(* Logix 5000 project; controller CHASKEY Emulate 5570 rev 30.12; software revision 30.00 *)

TASK MainTask (periodic, rate 3000 ms, priority 1, watchdog 5000 ms) : MainProgram

MODULES
   Local : Emulate 5570 (ICP 2, rev 30.12)
END_MODULES

VAR_GLOBAL   (* controller tags *)
   _SEC_P : BOOL;
   done : DINT;
   R_TRIG : FBD_ONESHOT;
   temp_var : DINT;
   test_array : DINT[20] := ([0] := 1, [1] := 2, [2] := 3, [3] := 4, [4] := 5, [5] := 6, [6] := 7, [7] := 8, [8] := 9, [9] := 10, [10] := 11, [11] := 12, [12] := 13, [13] := 14, [14] := 15, [15] := 16, [16] := 17, [17] := 18, [18] := 19, [19] := 20);
   TON : FBD_TIMER;
END_VAR

PROGRAM MainProgram   (* main routine MainRoutine *)
VAR
   Chaskey_128_i : DINT;
   Chaskey_a : DINT; {access None}
   Chaskey_BNum : DINT; {access None}
   Chaskey_i : DINT; {access None}
   Chaskey_IndexDiv : DINT;
   Chaskey_IndexMod : DINT;
   Chaskey_input_pi : DINT[4]; {access None}
   Chaskey_j : DINT; {access None}
   Chaskey_key : DINT[4]; {access None}
   Chaskey_L : DINT[4]; {access None}
   Chaskey_LastBlk : DINT[4];
   Chaskey_lb : DINT[16];
   Chaskey_Message : DINT[256]; {access None}
   Chaskey_mlen : DINT;
   Chaskey_MsgBitLen : DINT; {access None}
   Chaskey_MsgBlk : DINT[64];
   Chaskey_MsgBlkLen : DINT;
   Chaskey_per_i : DINT; {access None}
   Chaskey_round : DINT;
   Chaskey_subkey1_i : DINT; {access None}
   Chaskey_subkey2_i : DINT; {access None}
   Chaskey_subkey_1 : DINT[8];
   Chaskey_subkey_2 : DINT[8]; {access None}
   Chaskey_tag : DINT[4]; {access None}
   Chaskey_Temp : DINT; {access None}
   Chaskey_z : DINT;
   SCAN_CYCLE_TIME : DINT; {access None}
   test_i : DINT;
END_VAR

ROUTINE CHASKEY_128   (* structured text *)
   JSR(CHASKEY_Init);
   
   Chaskey_BNum:= Chaskey_MsgBitLen/128;
   
   if Chaskey_MsgBitLen mod 128 <>0 then
   	Chaskey_BNum:= Chaskey_BNum+1;
   end_if;
   
   
   for Chaskey_i:=0 to Chaskey_mlen by 1 do
   	Chaskey_MsgBlkLen:=Chaskey_mlen/4;
   	Chaskey_z:=Chaskey_i mod 4;
   	for Chaskey_j:=0 to 7 by 1 do
   		Chaskey_MsgBlk[Chaskey_MsgBlkLen].[Chaskey_z*8+Chaskey_j]:=Chaskey_Message[Chaskey_i].[Chaskey_j];
   	end_for;
   end_for;
   
   Chaskey_input_pi[3] := Chaskey_key[3];
   Chaskey_input_pi[2] := Chaskey_key[2] ;
   Chaskey_input_pi[1] := Chaskey_key[1] ;
   Chaskey_input_pi[0] := Chaskey_key[0] ;
   
   Chaskey_i:=0;
   if Chaskey_mlen<>0 then
   	while Chaskey_i < Chaskey_BNum-1 do
   		Chaskey_128_i:=Chaskey_i*4;
   		Chaskey_input_pi[3] := Chaskey_input_pi[3] XOR Chaskey_MsgBlk[Chaskey_128_i+3];
   		Chaskey_input_pi[2] := Chaskey_input_pi[2] XOR Chaskey_MsgBlk[Chaskey_128_i+2];
   		Chaskey_input_pi[1] := Chaskey_input_pi[1] XOR Chaskey_MsgBlk[Chaskey_128_i+1];
   		Chaskey_input_pi[0] := Chaskey_input_pi[0] XOR Chaskey_MsgBlk[Chaskey_128_i+0];
   		JSR(CHASKEY_Permutation);
   
   		if Chaskey_i>=Chaskey_BNum-2 then
   			Exit;
   		end_if;
   
   		Chaskey_i:=Chaskey_i +1;
   	end_while;
   end_if;
   
   
   if (Chaskey_mlen<>0) AND ((Chaskey_mlen & 15)=0) then
   	Chaskey_L[3] := Chaskey_subkey_1[3];
   	Chaskey_L[2] := Chaskey_subkey_1[2] ;
   	Chaskey_L[1] := Chaskey_subkey_1[1] ;
   	Chaskey_L[0] := Chaskey_subkey_1[0] ;
   	Chaskey_LastBlk[0]:=Chaskey_MsgBlk[0];
   	Chaskey_LastBlk[1]:=Chaskey_MsgBlk[1];
   	Chaskey_LastBlk[2]:=Chaskey_MsgBlk[2];
   	Chaskey_LastBlk[3]:=Chaskey_MsgBlk[3];
   else
   	Chaskey_L[3] := Chaskey_subkey_2[3];
   	Chaskey_L[2] := Chaskey_subkey_2[2] ;
   	Chaskey_L[1] := Chaskey_subkey_2[1] ;
   	Chaskey_L[0] := Chaskey_subkey_2[0] ;
   
   
   	Chaskey_IndexMod:= Chaskey_mlen mod 16;
   	Chaskey_IndexDiv:= (Chaskey_mlen/16)*16;
   	for Chaskey_j:=0 to Chaskey_IndexMod-1 by 1 do
   		Chaskey_lb[Chaskey_j]:=Chaskey_Message[Chaskey_IndexDiv+Chaskey_j];
   	end_for;
   	Chaskey_lb[Chaskey_IndexMod]:=1;
   	for Chaskey_j:=Chaskey_IndexMod+1 to 15 by 1 do
   		Chaskey_lb[Chaskey_j]:=0;
   	end_for;
   
   	//lastblock = (uint32_t*) lb;
   	Chaskey_LastBlk[0].0:=Chaskey_lb[0].0;
   	Chaskey_LastBlk[0].1:=Chaskey_lb[0].1;
   	Chaskey_LastBlk[0].2:=Chaskey_lb[0].2;
   	Chaskey_LastBlk[0].3:=Chaskey_lb[0].3;
   	Chaskey_LastBlk[0].4:=Chaskey_lb[0].4;
   	Chaskey_LastBlk[0].5:=Chaskey_lb[0].5;
   	Chaskey_LastBlk[0].6:=Chaskey_lb[0].6;
   	Chaskey_LastBlk[0].7:=Chaskey_lb[0].7;
   	Chaskey_LastBlk[0].8:=Chaskey_lb[1].0;
   	Chaskey_LastBlk[0].9:=Chaskey_lb[1].1;
   	Chaskey_LastBlk[0].10:=Chaskey_lb[1].2;
   	Chaskey_LastBlk[0].11:=Chaskey_lb[1].3;
   	Chaskey_LastBlk[0].12:=Chaskey_lb[1].4;
   	Chaskey_LastBlk[0].13:=Chaskey_lb[1].5;
   	Chaskey_LastBlk[0].14:=Chaskey_lb[1].6;
   	Chaskey_LastBlk[0].15:=Chaskey_lb[1].7;
   	Chaskey_LastBlk[0].16:=Chaskey_lb[2].0;
   	Chaskey_LastBlk[0].17:=Chaskey_lb[2].1;
   	Chaskey_LastBlk[0].18:=Chaskey_lb[2].2;
   	Chaskey_LastBlk[0].19:=Chaskey_lb[2].3;
   	Chaskey_LastBlk[0].20:=Chaskey_lb[2].4;
   	Chaskey_LastBlk[0].21:=Chaskey_lb[2].5;
   	Chaskey_LastBlk[0].22:=Chaskey_lb[2].6;
   	Chaskey_LastBlk[0].23:=Chaskey_lb[2].7;
   	Chaskey_LastBlk[0].24:=Chaskey_lb[3].0;
   	Chaskey_LastBlk[0].25:=Chaskey_lb[3].1;
   	Chaskey_LastBlk[0].26:=Chaskey_lb[3].2;
   	Chaskey_LastBlk[0].27:=Chaskey_lb[3].3;
   	Chaskey_LastBlk[0].28:=Chaskey_lb[3].4;
   	Chaskey_LastBlk[0].29:=Chaskey_lb[3].5;
   	Chaskey_LastBlk[0].30:=Chaskey_lb[3].6;
   	Chaskey_LastBlk[0].31:=Chaskey_lb[3].7;
   
   	Chaskey_LastBlk[1].0:=Chaskey_lb[4].0;
   	Chaskey_LastBlk[1].1:=Chaskey_lb[4].1;
   	Chaskey_LastBlk[1].2:=Chaskey_lb[4].2;
   	Chaskey_LastBlk[1].3:=Chaskey_lb[4].3;
   	Chaskey_LastBlk[1].4:=Chaskey_lb[4].4;
   	Chaskey_LastBlk[1].5:=Chaskey_lb[4].5;
   	Chaskey_LastBlk[1].6:=Chaskey_lb[4].6;
   	Chaskey_LastBlk[1].7:=Chaskey_lb[4].7;
   	Chaskey_LastBlk[1].8:=Chaskey_lb[5].0;
   	Chaskey_LastBlk[1].9:=Chaskey_lb[5].1;
   	Chaskey_LastBlk[1].10:=Chaskey_lb[5].2;
   	Chaskey_LastBlk[1].11:=Chaskey_lb[5].3;
   	Chaskey_LastBlk[1].12:=Chaskey_lb[5].4;
   	Chaskey_LastBlk[1].13:=Chaskey_lb[5].5;
   	Chaskey_LastBlk[1].14:=Chaskey_lb[5].6;
   	Chaskey_LastBlk[1].15:=Chaskey_lb[5].7;
   	Chaskey_LastBlk[1].16:=Chaskey_lb[6].0;
   	Chaskey_LastBlk[1].17:=Chaskey_lb[6].1;
   	Chaskey_LastBlk[1].18:=Chaskey_lb[6].2;
   	Chaskey_LastBlk[1].19:=Chaskey_lb[6].3;
   	Chaskey_LastBlk[1].20:=Chaskey_lb[6].4;
   	Chaskey_LastBlk[1].21:=Chaskey_lb[6].5;
   	Chaskey_LastBlk[1].22:=Chaskey_lb[6].6;
   	Chaskey_LastBlk[1].23:=Chaskey_lb[6].7;
   	Chaskey_LastBlk[1].24:=Chaskey_lb[7].0;
   	Chaskey_LastBlk[1].25:=Chaskey_lb[7].1;
   	Chaskey_LastBlk[1].26:=Chaskey_lb[7].2;
   	Chaskey_LastBlk[1].27:=Chaskey_lb[7].3;
   	Chaskey_LastBlk[1].28:=Chaskey_lb[7].4;
   	Chaskey_LastBlk[1].29:=Chaskey_lb[7].5;
   	Chaskey_LastBlk[1].30:=Chaskey_lb[7].6;
   	Chaskey_LastBlk[1].31:=Chaskey_lb[7].7;
   
   	Chaskey_LastBlk[2].0:=Chaskey_lb[8].0;
   	Chaskey_LastBlk[2].1:=Chaskey_lb[8].1;
   	Chaskey_LastBlk[2].2:=Chaskey_lb[8].2;
   	Chaskey_LastBlk[2].3:=Chaskey_lb[8].3;
   	Chaskey_LastBlk[2].4:=Chaskey_lb[8].4;
   	Chaskey_LastBlk[2].5:=Chaskey_lb[8].5;
   	Chaskey_LastBlk[2].6:=Chaskey_lb[8].6;
   	Chaskey_LastBlk[2].7:=Chaskey_lb[8].7;
   	Chaskey_LastBlk[2].8:=Chaskey_lb[9].0;
   	Chaskey_LastBlk[2].9:=Chaskey_lb[9].1;
   	Chaskey_LastBlk[2].10:=Chaskey_lb[9].2;
   	Chaskey_LastBlk[2].11:=Chaskey_lb[9].3;
   	Chaskey_LastBlk[2].12:=Chaskey_lb[9].4;
   	Chaskey_LastBlk[2].13:=Chaskey_lb[9].5;
   	Chaskey_LastBlk[2].14:=Chaskey_lb[9].6;
   	Chaskey_LastBlk[2].15:=Chaskey_lb[9].7;
   	Chaskey_LastBlk[2].16:=Chaskey_lb[10].0;
   	Chaskey_LastBlk[2].17:=Chaskey_lb[10].1;
   	Chaskey_LastBlk[2].18:=Chaskey_lb[10].2;
   	Chaskey_LastBlk[2].19:=Chaskey_lb[10].3;
   	Chaskey_LastBlk[2].20:=Chaskey_lb[10].4;
   	Chaskey_LastBlk[2].21:=Chaskey_lb[10].5;
   	Chaskey_LastBlk[2].22:=Chaskey_lb[10].6;
   	Chaskey_LastBlk[2].23:=Chaskey_lb[10].7;
   	Chaskey_LastBlk[2].24:=Chaskey_lb[11].0;
   	Chaskey_LastBlk[2].25:=Chaskey_lb[11].1;
   	Chaskey_LastBlk[2].26:=Chaskey_lb[11].2;
   	Chaskey_LastBlk[2].27:=Chaskey_lb[11].3;
   	Chaskey_LastBlk[2].28:=Chaskey_lb[11].4;
   	Chaskey_LastBlk[2].29:=Chaskey_lb[11].5;
   	Chaskey_LastBlk[2].30:=Chaskey_lb[11].6;
   	Chaskey_LastBlk[2].31:=Chaskey_lb[11].7;
   
   	Chaskey_LastBlk[3].0:=Chaskey_lb[12].0;
   	Chaskey_LastBlk[3].1:=Chaskey_lb[12].1;
   	Chaskey_LastBlk[3].2:=Chaskey_lb[12].2;
   	Chaskey_LastBlk[3].3:=Chaskey_lb[12].3;
   	Chaskey_LastBlk[3].4:=Chaskey_lb[12].4;
   	Chaskey_LastBlk[3].5:=Chaskey_lb[12].5;
   	Chaskey_LastBlk[3].6:=Chaskey_lb[12].6;
   	Chaskey_LastBlk[3].7:=Chaskey_lb[12].7;
   	Chaskey_LastBlk[3].8:=Chaskey_lb[13].0;
   	Chaskey_LastBlk[3].9:=Chaskey_lb[13].1;
   	Chaskey_LastBlk[3].10:=Chaskey_lb[13].2;
   	Chaskey_LastBlk[3].11:=Chaskey_lb[13].3;
   	Chaskey_LastBlk[3].12:=Chaskey_lb[13].4;
   	Chaskey_LastBlk[3].13:=Chaskey_lb[13].5;
   	Chaskey_LastBlk[3].14:=Chaskey_lb[13].6;
   	Chaskey_LastBlk[3].15:=Chaskey_lb[13].7;
   	Chaskey_LastBlk[3].16:=Chaskey_lb[14].0;
   	Chaskey_LastBlk[3].17:=Chaskey_lb[14].1;
   	Chaskey_LastBlk[3].18:=Chaskey_lb[14].2;
   	Chaskey_LastBlk[3].19:=Chaskey_lb[14].3;
   	Chaskey_LastBlk[3].20:=Chaskey_lb[14].4;
   	Chaskey_LastBlk[3].21:=Chaskey_lb[14].5;
   	Chaskey_LastBlk[3].22:=Chaskey_lb[14].6;
   	Chaskey_LastBlk[3].23:=Chaskey_lb[14].7;
   	Chaskey_LastBlk[3].24:=Chaskey_lb[15].0;
   	Chaskey_LastBlk[3].25:=Chaskey_lb[15].1;
   	Chaskey_LastBlk[3].26:=Chaskey_lb[15].2;
   	Chaskey_LastBlk[3].27:=Chaskey_lb[15].3;
   	Chaskey_LastBlk[3].28:=Chaskey_lb[15].4;
   	Chaskey_LastBlk[3].29:=Chaskey_lb[15].5;
   	Chaskey_LastBlk[3].30:=Chaskey_lb[15].6;
   	Chaskey_LastBlk[3].31:=Chaskey_lb[15].7;
   end_if;
   
   
   Chaskey_input_pi[3] := Chaskey_input_pi[3] XOR Chaskey_LastBlk[3] ;
   Chaskey_input_pi[2] := Chaskey_input_pi[2] XOR Chaskey_LastBlk[2] ;
   Chaskey_input_pi[1] := Chaskey_input_pi[1] XOR Chaskey_LastBlk[1] ;
   Chaskey_input_pi[0] := Chaskey_input_pi[0] XOR Chaskey_LastBlk[0] ;
   
   Chaskey_input_pi[3] := Chaskey_input_pi[3] XOR Chaskey_L[3] ;
   Chaskey_input_pi[2] := Chaskey_input_pi[2] XOR Chaskey_L[2] ;
   Chaskey_input_pi[1] := Chaskey_input_pi[1] XOR Chaskey_L[1] ;
   Chaskey_input_pi[0] := Chaskey_input_pi[0] XOR Chaskey_L[0] ;
   
   JSR(CHASKEY_Permutation);
   
   Chaskey_input_pi[3] := Chaskey_input_pi[3] XOR Chaskey_L[3] ;
   Chaskey_input_pi[2] := Chaskey_input_pi[2] XOR Chaskey_L[2] ;
   Chaskey_input_pi[1] := Chaskey_input_pi[1] XOR Chaskey_L[1] ;
   Chaskey_input_pi[0] := Chaskey_input_pi[0] XOR Chaskey_L[0] ;
   
   //////////////////////////////////////////////
   
   Chaskey_tag[3] := Chaskey_input_pi[3];
   Chaskey_tag[2] := Chaskey_input_pi[2];
   Chaskey_tag[1] := Chaskey_input_pi[1];
   Chaskey_tag[0] := Chaskey_input_pi[0];
   
   JSR(CHASKEY_ClearKey);
   
END_ROUTINE

ROUTINE CHASKEY_ClearKey   (* structured text *)
   
   Chaskey_key[0]:= 0;
   Chaskey_key[1]:= 0;
   Chaskey_key[2]:= 0;
   Chaskey_key[3]:= 0;
   
   
   Chaskey_subkey_1[0]:= 0;
   Chaskey_subkey_1[1]:= 0;
   Chaskey_subkey_1[2]:= 0;
   Chaskey_subkey_1[3]:= 0;
   
   Chaskey_subkey_2[0]:= 0;
   Chaskey_subkey_2[1]:= 0;
   Chaskey_subkey_2[2]:= 0;
   Chaskey_subkey_2[3]:= 0;
   
END_ROUTINE

ROUTINE CHASKEY_Init   (* structured text *)
    //key[3].31 is the MSB of the key, while key[0].0 is the LSB of the key
   (*Chaskey_key[0]:=0;
   Chaskey_key[1]:=17;
   Chaskey_key[2]:=34;
   Chaskey_key[3]:=51;*)
   
   Chaskey_key[0]:=857870592;
   Chaskey_key[1]:=2003195204;
   Chaskey_key[2]:=-1146447480;
   Chaskey_key[3]:=-1122868;
   
   Chaskey_tag[0] := 0;
   Chaskey_tag[1] := 0;
   Chaskey_tag[2] := 0;
   Chaskey_tag[3] := 0;
   
   //Initialize subkey_1[] and subkey_2[]
   Chaskey_subkey_1[0] := 1715741319;
   Chaskey_subkey_1[1] := -288576888;
   Chaskey_subkey_1[2] := 2002070336;
   Chaskey_subkey_1[3] := -2245735;
   
   Chaskey_subkey_2[0] := -863484535;
   Chaskey_subkey_2[1] := -577153776;
   Chaskey_subkey_2[2] := -290822623;
   Chaskey_subkey_2[3] := -4491470;
   
   
   
END_ROUTINE

ROUTINE CHASKEY_Permutation   (* structured text *)
   
   for Chaskey_per_i:=0 to Chaskey_round by 1 do
   
   
   	Chaskey_input_pi[0]:= Chaskey_input_pi[0] + Chaskey_input_pi[1];
   
   	Chaskey_a:=Chaskey_input_pi[1];  //v1 <<< 5
   	Chaskey_Temp:=0;
   	//left shift Chaskey_b=5 bits
   	Chaskey_Temp.5:=Chaskey_a.0;
   	Chaskey_Temp.6:=Chaskey_a.1;
   	Chaskey_Temp.7:=Chaskey_a.2;
   	Chaskey_Temp.8:=Chaskey_a.3;
   	Chaskey_Temp.9:=Chaskey_a.4;
   	Chaskey_Temp.10:=Chaskey_a.5;
   	Chaskey_Temp.11:=Chaskey_a.6;
   	Chaskey_Temp.12:=Chaskey_a.7;
   	Chaskey_Temp.13:=Chaskey_a.8;
   	Chaskey_Temp.14:=Chaskey_a.9;
   	Chaskey_Temp.15:=Chaskey_a.10;
   	Chaskey_Temp.16:=Chaskey_a.11;
   	Chaskey_Temp.17:=Chaskey_a.12;
   	Chaskey_Temp.18:=Chaskey_a.13;
   	Chaskey_Temp.19:=Chaskey_a.14;
   	Chaskey_Temp.20:=Chaskey_a.15;
   	Chaskey_Temp.21:=Chaskey_a.16;
   	Chaskey_Temp.22:=Chaskey_a.17;
   	Chaskey_Temp.23:=Chaskey_a.18;
   	Chaskey_Temp.24:=Chaskey_a.19;
   	Chaskey_Temp.25:=Chaskey_a.20;
   	Chaskey_Temp.26:=Chaskey_a.21;
   	Chaskey_Temp.27:=Chaskey_a.22;
   	Chaskey_Temp.28:=Chaskey_a.23;
   	Chaskey_Temp.29:=Chaskey_a.24;
   	Chaskey_Temp.30:=Chaskey_a.25;
   	Chaskey_Temp.31:=Chaskey_a.26;
   	Chaskey_Temp.0:=Chaskey_a.27;
   	Chaskey_Temp.1:=Chaskey_a.28;
   	Chaskey_Temp.2:=Chaskey_a.29;
   	Chaskey_Temp.3:=Chaskey_a.30;
   	Chaskey_Temp.4:=Chaskey_a.31;
   	Chaskey_input_pi[1]:=Chaskey_Temp;
   
   	Chaskey_input_pi[1]:=Chaskey_input_pi[1] XOR Chaskey_input_pi[0];
   
   
   	Chaskey_a:=Chaskey_input_pi[0];  // <<< 16
   	Chaskey_Temp:=0;
   	//left shift Chaskey_b=16 bits
   	Chaskey_Temp.16:=Chaskey_a.0;
   	Chaskey_Temp.17:=Chaskey_a.1;
   	Chaskey_Temp.18:=Chaskey_a.2;
   	Chaskey_Temp.19:=Chaskey_a.3;
   	Chaskey_Temp.20:=Chaskey_a.4;
   	Chaskey_Temp.21:=Chaskey_a.5;
   	Chaskey_Temp.22:=Chaskey_a.6;
   	Chaskey_Temp.23:=Chaskey_a.7;
   	Chaskey_Temp.24:=Chaskey_a.8;
   	Chaskey_Temp.25:=Chaskey_a.9;
   	Chaskey_Temp.26:=Chaskey_a.10;
   	Chaskey_Temp.27:=Chaskey_a.11;
   	Chaskey_Temp.28:=Chaskey_a.12;
   	Chaskey_Temp.29:=Chaskey_a.13;
   	Chaskey_Temp.30:=Chaskey_a.14;
   	Chaskey_Temp.31:=Chaskey_a.15;
   	Chaskey_Temp.0:=Chaskey_a.16;
   	Chaskey_Temp.1:=Chaskey_a.17;
   	Chaskey_Temp.2:=Chaskey_a.18;
   	Chaskey_Temp.3:=Chaskey_a.19;
   	Chaskey_Temp.4:=Chaskey_a.20;
   	Chaskey_Temp.5:=Chaskey_a.21;
   	Chaskey_Temp.6:=Chaskey_a.22;
   	Chaskey_Temp.7:=Chaskey_a.23;
   	Chaskey_Temp.8:=Chaskey_a.24;
   	Chaskey_Temp.9:=Chaskey_a.25;
   	Chaskey_Temp.10:=Chaskey_a.26;
   	Chaskey_Temp.11:=Chaskey_a.27;
   	Chaskey_Temp.12:=Chaskey_a.28;
   	Chaskey_Temp.13:=Chaskey_a.29;
   	Chaskey_Temp.14:=Chaskey_a.30;
   	Chaskey_Temp.15:=Chaskey_a.31;
   	Chaskey_input_pi[0]:=Chaskey_Temp;
   
   
       Chaskey_input_pi[2]:= Chaskey_input_pi[2] + Chaskey_input_pi[3];
   
   
   	Chaskey_a:=Chaskey_input_pi[3];  // <<< 8
   	Chaskey_Temp:=0;
   	//left shift Chaskey_b=8 bits
   	Chaskey_Temp.8:=Chaskey_a.0;
   	Chaskey_Temp.9:=Chaskey_a.1;
   	Chaskey_Temp.10:=Chaskey_a.2;
   	Chaskey_Temp.11:=Chaskey_a.3;
   	Chaskey_Temp.12:=Chaskey_a.4;
   	Chaskey_Temp.13:=Chaskey_a.5;
   	Chaskey_Temp.14:=Chaskey_a.6;
   	Chaskey_Temp.15:=Chaskey_a.7;
   	Chaskey_Temp.16:=Chaskey_a.8;
   	Chaskey_Temp.17:=Chaskey_a.9;
   	Chaskey_Temp.18:=Chaskey_a.10;
   	Chaskey_Temp.19:=Chaskey_a.11;
   	Chaskey_Temp.20:=Chaskey_a.12;
   	Chaskey_Temp.21:=Chaskey_a.13;
   	Chaskey_Temp.22:=Chaskey_a.14;
   	Chaskey_Temp.23:=Chaskey_a.15;
   	Chaskey_Temp.24:=Chaskey_a.16;
   	Chaskey_Temp.25:=Chaskey_a.17;
   	Chaskey_Temp.26:=Chaskey_a.18;
   	Chaskey_Temp.27:=Chaskey_a.19;
   	Chaskey_Temp.28:=Chaskey_a.20;
   	Chaskey_Temp.29:=Chaskey_a.21;
   	Chaskey_Temp.30:=Chaskey_a.22;
   	Chaskey_Temp.31:=Chaskey_a.23;
   	Chaskey_Temp.0:=Chaskey_a.24;
   	Chaskey_Temp.1:=Chaskey_a.25;
   	Chaskey_Temp.2:=Chaskey_a.26;
   	Chaskey_Temp.3:=Chaskey_a.27;
   	Chaskey_Temp.4:=Chaskey_a.28;
   	Chaskey_Temp.5:=Chaskey_a.29;
   	Chaskey_Temp.6:=Chaskey_a.30;
   	Chaskey_Temp.7:=Chaskey_a.31;
   	Chaskey_input_pi[3]:=Chaskey_Temp;
   
   	Chaskey_input_pi[3]:=Chaskey_input_pi[3] XOR Chaskey_input_pi[2];
   
   
   
   	Chaskey_input_pi[0]:= Chaskey_input_pi[0] + Chaskey_input_pi[3];
   
   	Chaskey_a:=Chaskey_input_pi[3];  //<<< 13
   	Chaskey_Temp:=0;
   	//left shift Chaskey_b=13 bits
   	Chaskey_Temp.13:=Chaskey_a.0;
   	Chaskey_Temp.14:=Chaskey_a.1;
   	Chaskey_Temp.15:=Chaskey_a.2;
   	Chaskey_Temp.16:=Chaskey_a.3;
   	Chaskey_Temp.17:=Chaskey_a.4;
   	Chaskey_Temp.18:=Chaskey_a.5;
   	Chaskey_Temp.19:=Chaskey_a.6;
   	Chaskey_Temp.20:=Chaskey_a.7;
   	Chaskey_Temp.21:=Chaskey_a.8;
   	Chaskey_Temp.22:=Chaskey_a.9;
   	Chaskey_Temp.23:=Chaskey_a.10;
   	Chaskey_Temp.24:=Chaskey_a.11;
   	Chaskey_Temp.25:=Chaskey_a.12;
   	Chaskey_Temp.26:=Chaskey_a.13;
   	Chaskey_Temp.27:=Chaskey_a.14;
   	Chaskey_Temp.28:=Chaskey_a.15;
   	Chaskey_Temp.29:=Chaskey_a.16;
   	Chaskey_Temp.30:=Chaskey_a.17;
   	Chaskey_Temp.31:=Chaskey_a.18;
   	Chaskey_Temp.0:=Chaskey_a.19;
   	Chaskey_Temp.1:=Chaskey_a.20;
   	Chaskey_Temp.2:=Chaskey_a.21;
   	Chaskey_Temp.3:=Chaskey_a.22;
   	Chaskey_Temp.4:=Chaskey_a.23;
   	Chaskey_Temp.5:=Chaskey_a.24;
   	Chaskey_Temp.6:=Chaskey_a.25;
   	Chaskey_Temp.7:=Chaskey_a.26;
   	Chaskey_Temp.8:=Chaskey_a.27;
   	Chaskey_Temp.9:=Chaskey_a.28;
   	Chaskey_Temp.10:=Chaskey_a.29;
   	Chaskey_Temp.11:=Chaskey_a.30;
   	Chaskey_Temp.12:=Chaskey_a.31;
   	Chaskey_input_pi[3]:=Chaskey_Temp;
   
   	Chaskey_input_pi[3]:=Chaskey_input_pi[3] XOR Chaskey_input_pi[0];
   
   
   	Chaskey_input_pi[2]:=  Chaskey_input_pi[2] + Chaskey_input_pi[1];
   
   	Chaskey_a:=Chaskey_input_pi[1]; //<<< 7
   	Chaskey_Temp:=0;
   	//left shift Chaskey_b=7 bits
   	Chaskey_Temp.7:=Chaskey_a.0;
   	Chaskey_Temp.8:=Chaskey_a.1;
   	Chaskey_Temp.9:=Chaskey_a.2;
   	Chaskey_Temp.10:=Chaskey_a.3;
   	Chaskey_Temp.11:=Chaskey_a.4;
   	Chaskey_Temp.12:=Chaskey_a.5;
   	Chaskey_Temp.13:=Chaskey_a.6;
   	Chaskey_Temp.14:=Chaskey_a.7;
   	Chaskey_Temp.15:=Chaskey_a.8;
   	Chaskey_Temp.16:=Chaskey_a.9;
   	Chaskey_Temp.17:=Chaskey_a.10;
   	Chaskey_Temp.18:=Chaskey_a.11;
   	Chaskey_Temp.19:=Chaskey_a.12;
   	Chaskey_Temp.20:=Chaskey_a.13;
   	Chaskey_Temp.21:=Chaskey_a.14;
   	Chaskey_Temp.22:=Chaskey_a.15;
   	Chaskey_Temp.23:=Chaskey_a.16;
   	Chaskey_Temp.24:=Chaskey_a.17;
   	Chaskey_Temp.25:=Chaskey_a.18;
   	Chaskey_Temp.26:=Chaskey_a.19;
   	Chaskey_Temp.27:=Chaskey_a.20;
   	Chaskey_Temp.28:=Chaskey_a.21;
   	Chaskey_Temp.29:=Chaskey_a.22;
   	Chaskey_Temp.30:=Chaskey_a.23;
   	Chaskey_Temp.31:=Chaskey_a.24;
   	Chaskey_Temp.0:=Chaskey_a.25;
   	Chaskey_Temp.1:=Chaskey_a.26;
   	Chaskey_Temp.2:=Chaskey_a.27;
   	Chaskey_Temp.3:=Chaskey_a.28;
   	Chaskey_Temp.4:=Chaskey_a.29;
   	Chaskey_Temp.5:=Chaskey_a.30;
   	Chaskey_Temp.6:=Chaskey_a.31;
   	Chaskey_input_pi[1]:=Chaskey_Temp;
   
   	Chaskey_input_pi[1]:=Chaskey_input_pi[1] XOR Chaskey_input_pi[2];
   
   
   	Chaskey_a:=Chaskey_input_pi[2];   //<<< 16
   	Chaskey_Temp:=0;
   	//left shift Chaskey_b=16 bits
   	Chaskey_Temp.16:=Chaskey_a.0;
   	Chaskey_Temp.17:=Chaskey_a.1;
   	Chaskey_Temp.18:=Chaskey_a.2;
   	Chaskey_Temp.19:=Chaskey_a.3;
   	Chaskey_Temp.20:=Chaskey_a.4;
   	Chaskey_Temp.21:=Chaskey_a.5;
   	Chaskey_Temp.22:=Chaskey_a.6;
   	Chaskey_Temp.23:=Chaskey_a.7;
   	Chaskey_Temp.24:=Chaskey_a.8;
   	Chaskey_Temp.25:=Chaskey_a.9;
   	Chaskey_Temp.26:=Chaskey_a.10;
   	Chaskey_Temp.27:=Chaskey_a.11;
   	Chaskey_Temp.28:=Chaskey_a.12;
   	Chaskey_Temp.29:=Chaskey_a.13;
   	Chaskey_Temp.30:=Chaskey_a.14;
   	Chaskey_Temp.31:=Chaskey_a.15;
   	Chaskey_Temp.0:=Chaskey_a.16;
   	Chaskey_Temp.1:=Chaskey_a.17;
   	Chaskey_Temp.2:=Chaskey_a.18;
   	Chaskey_Temp.3:=Chaskey_a.19;
   	Chaskey_Temp.4:=Chaskey_a.20;
   	Chaskey_Temp.5:=Chaskey_a.21;
   	Chaskey_Temp.6:=Chaskey_a.22;
   	Chaskey_Temp.7:=Chaskey_a.23;
   	Chaskey_Temp.8:=Chaskey_a.24;
   	Chaskey_Temp.9:=Chaskey_a.25;
   	Chaskey_Temp.10:=Chaskey_a.26;
   	Chaskey_Temp.11:=Chaskey_a.27;
   	Chaskey_Temp.12:=Chaskey_a.28;
   	Chaskey_Temp.13:=Chaskey_a.29;
   	Chaskey_Temp.14:=Chaskey_a.30;
   	Chaskey_Temp.15:=Chaskey_a.31;
   	Chaskey_input_pi[2]:=Chaskey_Temp;
   end_for;
   
   
END_ROUTINE

ROUTINE CHASKEY_Test   (* structured text *)
   if S:FS then
   
   (*	Chaskey_input_pi[0]:= -2054128804;
   	Chaskey_input_pi[1]:= -1998792764;
   	Chaskey_input_pi[2]:= 1871086030;
   	Chaskey_input_pi[3]:= 1068001685;*)
   
   (* //test permutation
    	Chaskey_round:=11;
   	Chaskey_input_pi[0]:= 857870592;
   	Chaskey_input_pi[1]:= 2003195204;
   	Chaskey_input_pi[2]:= -1146447480;
   	Chaskey_input_pi[3]:= -1122868;
   
       Chaskey_LastBlk[0]:= 1;
   	Chaskey_LastBlk[1]:= 0;
   	Chaskey_LastBlk[2]:= 0;
   	Chaskey_LastBlk[3]:= 0;
   	JSR(CHASKEY_128);  *)
   
   	Chaskey_mlen:=0;
   	Chaskey_MsgBitLen:=(Chaskey_mlen+1)*8; //bit length of message
   
   	for test_i:=0 to Chaskey_mlen by 1 do
      		Chaskey_Message[test_i]:= test_i;
   	end_for;
   
   	Chaskey_round:=11;
   	JSR(CHASKEY_128);
   
   end_if;
END_ROUTINE

ROUTINE MainRoutine   (* ladder *)
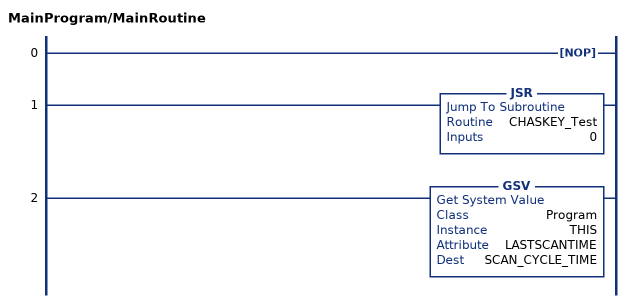
   0: NOP();
   1: JSR(CHASKEY_Test,0);
   2: GSV(Program,THIS,LASTSCANTIME,SCAN_CYCLE_TIME);
END_ROUTINE
END_PROGRAM
